(* IEC 61131-3 sources: Summary-ETFA22/ahorn/test/benchmark/dissertation/augmentation/presentation/S, 1 file *)

(* ---- S.st ---- *)
PROGRAM P
VAR_INPUT
    x : INT;
END_VAR
VAR
    y : INT;
END_VAR
VAR_OUTPUT
    z : BOOL;
END_VAR
    y := change(x, x + 1);
    IF y > 1 THEN
        z := TRUE;
    ELSE
        z := FALSE;
    END_IF;
END_PROGRAM
